(* Logix 5000 project; controller STAT 1756-L72 rev 20.12; software revision 20.04 *)

TASK IBT (periodic, rate 50 ms, priority 10, watchdog 200 ms) : ibt, stock, BASSIN
TASK MainTask (event, rate 200 ms, priority 15, watchdog 500 ms) : MainProgram

MODULES
   Local : 1756-L72 (ICP 0, rev 20.12)
        arm1_flex:0:I.1   // NIV_MID_VLOK1
        arm1_flex:0:I.2   // NIV_LAAG_VLOK1
        arm1_flex:0:I.4   // NIV_MID_VLOK2 FLOCULANT
        arm1_flex:0:I.5   // NIV_LAAG_VLOK2
        arm1_flex:0:I.6   // FC EV3
        arm1_flex:0:I.7   // FC EV3
        arm1_flex:0:I.12   // FLOW SWITCH PM4
        arm1_flex:0:I.13   // FLOW SWITCH PM2
        arm1_flex:0:I.14   // FLOW SWITCH PM3
        arm1_flex:0:I.15   // FLOW SWITCH PM4
        armstat_flex1:1:I.1   // CL3 MANU/AUTO
        armstat_flex1:4:O.0   // L P11 RUN
        armstat_flex1:4:O.1   // L P11 STOP/def
        armstat_flex1:4:O.2   // L P12 RUN
        armstat_flex1:4:O.3   // L P12 STOP/def
        armstat_flex1:4:O.4   // RES
        armstat_flex1:4:O.5   // RES
        armstat_flex1:4:O.6   // RES
        armstat_flex1:4:O.7   // RES
        armstat_flex1:4:O.8   // L P13 RUN
        armstat_flex1:4:O.9   // L P13 STOP/def
        armstat_flex1:4:O.10   // L P14 RUN
        armstat_flex1:4:O.11   // L P14 STOP/def
        armstat_flex1:4:O.12   // RES
        armstat_flex1:4:O.13   // RES
        armstat_flex1:4:O.14   // RES
        armstat_flex1:4:O.15   // RES
        armstat_flex1:0:I.1   // CL2 MANU/AUTO
        arm1_flex:1:I.0   // STFA11 EV1 BOVEN OPEN
        arm1_flex:1:I.1   // STFA11 EV1 BOVEN TOE
        arm1_flex:1:I.2   // STFA11 EV1 ONDER OPEN
        arm1_flex:1:I.3   // STFA11 EV1 ONDER TOE
        arm1_flex:1:I.4   // STFA12 EV1 BOVEN OPEN
        arm1_flex:1:I.5   // STFA12 EV1 BOVEN TOE
        arm1_flex:1:I.6   // STFA12 EV1 ONDER OPEN
        arm1_flex:1:I.7   // STFA12 EV1 ONDER TOE
        armstat_flex1:5:O.0   // L P15 RUN
        armstat_flex1:5:O.1   // L P15 STOP/def
        armstat_flex1:5:O.2   // L P16 RUN
        armstat_flex1:5:O.3   // L P16 STOP/def
        armstat_flex1:5:O.4   // RES
        armstat_flex1:5:O.5   // RES
        armstat_flex1:5:O.6   // RES
        armstat_flex1:5:O.7   // RES
        armstat_flex1:5:O.10   // RES
        armstat_flex1:5:O.11   // RES
        armstat_flex1:5:O.12   // RES
        armstat_flex1:5:O.13   // RES
        armstat_flex1:5:O.14   // RES
        armstat_flex1:5:O.15   // RES
        armstat_flex1:2:I.1   // CL4 MANU/AUTO
      usine : 1756-ENBT (Ethernet 192.168.3.162, ICP 1, rev 5.1)
         L1_usine : 1756-ENBT (Ethernet 192.168.3.159, rev 5.1)
            L1 : 1756-L72 (ICP 5, rev 20.1, $f88beb9a$ RPI 250 ms)
         EtherNet_Bridge : 1756-ENBT (Ethernet 192.168.3.150, rev 4.3)
            wkk : vendor 1 type 14 code 92 (ICP 2, rev 20.1, $435658c3$ RPI 20 ms)
         L2_usine : 1756-EN2T (Ethernet 192.168.3.163, rev 3.1)
            @63fa20a3@:Partner : vendor 1 type 14 code 146 (ICP 5, rev 20.1)
            L2PROCESS : vendor 1 type 14 code 147 (ICP 4, rev 20.1, $7ef97ec5$ RPI 20 ms)
         L3_usine : 1756-EN2T (Ethernet 192.168.3.161, rev 3.1)
            L3 : vendor 1 type 14 code 92 (ICP 0, rev 20.1, $abc03147$ RPI 250 ms)
      IO : 1756-ENBT (ICP 2, Ethernet 192.168.1.1, rev 6.4)
         arm1_flex : 1794-AENTR (Ethernet 192.168.1.8, rev 1.1, Output RPI 20 ms)
            I1_2 : 1794-IB16 (Flex 1, rev 1.1)
            I1_1 : 1794-IB16 (Flex 0, rev 1.1)
            I1_5 : 1794-IB16 (Flex 5, rev 1.1)
            O1_6 : vendor 1 type 7 code 35 (Flex 6, rev 1.1)
            N20 : vendor 1 type 10 code 31 (Flex 2, rev 1.1, Output RPI 80 ms)
            N21 : vendor 1 type 10 code 31 (Flex 3, rev 1.1, Output RPI 80 ms)
            N22 : vendor 1 type 10 code 31 (Flex 4, rev 1.1, Output RPI 80 ms)
         armstat_flex2 : 1794-AENTR (Ethernet 192.168.1.7, rev 1.1, Output RPI 20 ms)
            future : vendor 1 type 10 code 30 (Flex 1, rev 1.1, Input RPI 80 ms)
            N19_0 : vendor 1 type 10 code 30 (Flex 0, rev 1.1, Input RPI 80 ms)
         armPmp_flex1 : 1794-AENTR (Ethernet 192.168.1.5, rev 1.1, Output RPI 20 ms)
            I1_10 : 1794-IB16 (Flex 2, rev 1.1)
            I1_9 : 1794-IB16 (Flex 1, rev 1.1)
            O1_11 : vendor 1 type 7 code 35 (Flex 3, rev 1.1)
            I1_8 : 1794-IB16 (Flex 0, rev 1.1)
            O1_12 : vendor 1 type 7 code 35 (Flex 4, rev 1.1)
            N24 : vendor 1 type 10 code 31 (Flex 6, rev 1.1, Output RPI 80 ms)
            N23 : vendor 1 type 10 code 30 (Flex 5, rev 1.1, Input RPI 80 ms)
         armstat_flex1 : 1794-AENTR (Ethernet 192.168.1.6, rev 1.1, Output RPI 20 ms)
            I1_17 : 1794-IB16 (Flex 1, rev 1.1)
            O1_21 : vendor 1 type 7 code 35 (Flex 5, rev 1.1)
            I1_19 : 1794-IB16 (Flex 3, rev 1.1)
            I1_16 : 1794-IB16 (Flex 0, rev 1.1)
            I1_18 : 1794-IB16 (Flex 2, rev 1.1)
            O1_20 : vendor 1 type 7 code 35 (Flex 4, rev 1.1)
            N7_0 : vendor 1 type 10 code 30 (Flex 6, rev 1.1, Input RPI 80 ms)
         switch : vendor 1 type 12 code 238 (Ethernet 192.168.1.20, rev 3.1, StandardDataDriven RPI 1000 ms)
         bassin : vendor 1 type 12 code 228 (Ethernet 192.168.1.11, rev 1.1)
            bas_I_01 : vendor 1 type 116 code 6 (SLCChassis 1, rev 1.1, StandardDataDriven RPI 200 ms)
                 bassin:1:I.DATA.0   // fc vanne venturi ouverte vers venturi
                 bassin:1:I.DATA.1   // fc vanne venturi fermée vers bassin
                 bassin:1:I.DATA.2   // fc vanne PH bac ouverte
                 bassin:1:I.DATA.3   // fc vanne PH bac fermée
                 bassin:1:I.DATA.4   // fc vanne Neutral ouverte
                 bassin:1:I.DATA.5   // fc vanne Neutral fermée
                 bassin:1:I.DATA.6   // defaut ultima pmp renvoi 1
                 bassin:1:I.DATA.7   // defaut ultima pmp renvoi 2
                 bassin:1:I.DATA.8   // sélecteur local pmp renvoi 1
                 bassin:1:I.DATA.9   // Bp M/A loc pmp renvoi 1
                 bassin:1:I.DATA.10   // sélecteur local pmp renvoi 2
                 bassin:1:I.DATA.11   // Bp M/A loc pmp renvoi 2
                 bassin:1:I.DATA.12   // Bp M/A dist pmp renvoi 1
                 bassin:1:I.DATA.13   // Bp M/A dist pmp renvoi 2
                 bassin:1:I.DATA.14   // présence pmp renvoi 1
                 bassin:1:I.DATA.15   // présence pmp renvoi 2
                 bassin:1:I.DATA.16   // ready drive pmp acide nautral
                 bassin:1:I.DATA.17   // ready drive pmp base neutral
                 bassin:1:I.DATA.18   // selecteur fermer vanne
                 bassin:1:I.DATA.19   // reserve
                 bassin:1:I.DATA.20   // reserve
                 bassin:1:I.DATA.21   // reserve
                 bassin:1:I.DATA.22   // reserve
                 bassin:1:I.DATA.23   // reserve
                 bassin:1:I.DATA.24   // reserve
                 bassin:1:I.DATA.25   // reserve
                 bassin:1:I.DATA.26   // reserve
                 bassin:1:I.DATA.27   // reserve
                 bassin:1:I.DATA.28   // reserve
                 bassin:1:I.DATA.29   // reserve
                 bassin:1:I.DATA.30   // reserve
                 bassin:1:I.DATA.31   // reserve
            bas_AI_03 : vendor 1 type 117 code 6 (SLCChassis 3, rev 1.1, StandardDataDriven RPI 200 ms)
            bas_O_02 : vendor 1 type 116 code 30 (SLCChassis 2, rev 1.1, StandardDataDriven RPI 200 ms)
                 bassin:2:O.POINT_11   // pmp acide
                 bassin:2:O.POINT_12   // ajout base
                 bassin:2:O.DATA.0   // marche pmp 1 renvoi
                 bassin:2:O.DATA.1   // marche pmp 2 renvoi
                 bassin:2:O.DATA.2   // ouverturre vanne venturi
                 bassin:2:O.DATA.3   // lampe M/A loc pmp renvoi 1
                 bassin:2:O.DATA.4   // lampe M/A loc pmp renvoi 2
                 bassin:2:O.DATA.5   // lampe M/A dist pmp renvoi 1
                 bassin:2:O.DATA.6   // lampe M/A dist pmp renvoi 2
                 bassin:2:O.DATA.7   // colone lumineuse bleu discord. vanne manu
                 bassin:2:O.DATA.8   // colone lumineuse niveau bas bassin
                 bassin:2:O.DATA.9   // colone lumineuse defaut pompe renvoi
                 bassin:2:O.DATA.10   // colone lumineuse rouge
                 bassin:2:O.DATA.11   // M/A drive PMP acide neutral
                 bassin:2:O.DATA.12   // M/A drive PMP base neutral
                 bassin:2:O.DATA.13   // reserve
                 bassin:2:O.DATA.14   // reserve
                 bassin:2:O.DATA.15   // reserve
                 bassin:2:O.DATA.16   // reserve
                 bassin:2:O.DATA.17   // reserve
                 bassin:2:O.DATA.18   // reserve
                 bassin:2:O.DATA.19   // reserve
                 bassin:2:O.DATA.20   // reserve
                 bassin:2:O.DATA.21   // reserve
                 bassin:2:O.DATA.22   // reserve
                 bassin:2:O.DATA.23   // reserve
                 bassin:2:O.DATA.24   // reserve
                 bassin:2:O.DATA.25   // reserve
                 bassin:2:O.DATA.26   // reserve
                 bassin:2:O.DATA.27   // reserve
                 bassin:2:O.DATA.28   // reserve
                 bassin:2:O.DATA.29   // reserve
                 bassin:2:O.DATA.30   // reserve
                 bassin:2:O.DATA.31   // reserve
            bas_AO_04 : vendor 1 type 117 code 11 (SLCChassis 4, rev 1.1, StandardDataDriven RPI 200 ms)
                 bassin:4:O.CHANNEL_0_OUTPUT   // consigne position vanne renvoi
                 bassin:4:O.CHANNEL_1_OUTPUT   // consigne vitesse pmp acide neutral
                 bassin:4:O.CHANNEL_2_OUTPUT   // consigne vitesse pmp base neutral
         Lancy_R2 : vendor 1 type 12 code 228 (Ethernet 192.168.1.14, rev 1.1)
            lancy_R2_O2 : vendor 1 type 116 code 23 (SLCChassis 2, rev 1.1, StandardDataDriven RPI 200 ms)
                 Lancy_R2:2:O.DATA.0   // drum wash frequency. duration timer panel+G116
                 Lancy_R2:2:O.DATA.1   // surge tank T150 overflow shut off valve
                 Lancy_R2:2:O.DATA.2   // AV 147 open
                 Lancy_R2:2:O.DATA.3   // AV 147 close
                 Lancy_R2:2:O.DATA.4   // caustic supply P190
                 Lancy_R2:2:O.DATA.5   // P190 on
                 Lancy_R2:2:O.DATA.6   // ST VA7 Vanne eau rinçage
                 Lancy_R2:2:O.DATA.7   // ST VA7 Vanne eau rinçage
                 Lancy_R2:2:O.POINT_0   // drum wash frequency. duration timer panel+G116
                 Lancy_R2:2:O.POINT_1   // surge tank T150 overflow shut off valve
                 Lancy_R2:2:O.POINT_2   // AV 147 open
                 Lancy_R2:2:O.POINT_3   // AV 147 close
                 Lancy_R2:2:O.POINT_4   // caustic supply P190
                 Lancy_R2:2:O.POINT_5   // P190 on
                 Lancy_R2:2:O.POINT_6   // ST VA7 Vanne eau rinçage
                 Lancy_R2:2:O.POINT_7   // ST VA7 Vanne eau rinçage
            lancy_R2_O6 : vendor 1 type 116 code 23 (SLCChassis 6, rev 1.1, StandardDataDriven RPI 200 ms)
                 Lancy_R2:6:O.DATA.0   // AV 330 closed
                 Lancy_R2:6:O.DATA.1   // alarm horn
                 Lancy_R2:6:O.DATA.2   // L1 high level
                 Lancy_R2:6:O.DATA.3   // L1 low level
                 Lancy_R2:6:O.DATA.4   // L2 high level
                 Lancy_R2:6:O.DATA.5   // L2 low level
                 Lancy_R2:6:O.DATA.6   // L3 high level
                 Lancy_R2:6:O.DATA.7   // L3 low level
                 Lancy_R2:6:O.POINT_0   // AV 330 closed
                 Lancy_R2:6:O.POINT_1   // alarm horn
                 Lancy_R2:6:O.POINT_2   // L1 high level
                 Lancy_R2:6:O.POINT_3   // L1 low level
                 Lancy_R2:6:O.POINT_4   // L2 high level
                 Lancy_R2:6:O.POINT_5   // L2 low level
                 Lancy_R2:6:O.POINT_6   // L3 high level
                 Lancy_R2:6:O.POINT_7   // L3 low level
            lancy_R2_O9 : vendor 1 type 116 code 23 (SLCChassis 9, rev 1.1, StandardDataDriven RPI 200 ms)
                 Lancy_R2:9:O.DATA.0   // cloudy filtrate P240 overcurrent
                 Lancy_R2:9:O.DATA.1   // rotary drum F200 overcurrent
                 Lancy_R2:9:O.DATA.2   // vacuum pump P250 overcurrent
                 Lancy_R2:9:O.DATA.3   // clear filtrate pump failure
                 Lancy_R2:9:O.DATA.4   // cloudy filtrate pump failure
                 Lancy_R2:9:O.DATA.5   // filtrate lift station pump failure
                 Lancy_R2:9:O.DATA.6   // regenerate caustic avalaible holding tank
                 Lancy_R2:9:O.DATA.7   // System high level alarm
                 Lancy_R2:9:O.POINT_0   // cloudy filtrate P240 overcurrent
                 Lancy_R2:9:O.POINT_1   // rotary drum F200 overcurrent
                 Lancy_R2:9:O.POINT_2   // vacuum pump P250 overcurrent
                 Lancy_R2:9:O.POINT_3   // clear filtrate pump failure
                 Lancy_R2:9:O.POINT_4   // cloudy filtrate pump failure
                 Lancy_R2:9:O.POINT_5   // filtrate lift station pump failure
                 Lancy_R2:9:O.POINT_6   // regenerate caustic avalaible holding tank
                 Lancy_R2:9:O.POINT_7   // System high level alarm
            lancy_R2_O7 : vendor 1 type 116 code 23 (SLCChassis 7, rev 1.1, StandardDataDriven RPI 200 ms)
                 Lancy_R2:7:O.DATA.0   // holding tank T130 high level
                 Lancy_R2:7:O.DATA.1   // filtrate lift station T160 high level
                 Lancy_R2:7:O.DATA.2   // clear filtrate receiver T260 high level
                 Lancy_R2:7:O.DATA.3   // cloudy filtrate receiver T270 high level
                 Lancy_R2:7:O.DATA.4   // vacuum pump sunction line high level
                 Lancy_R2:7:O.DATA.5   // reactor tank T100 high level
                 Lancy_R2:7:O.DATA.6   // reactor tank T100 low level
                 Lancy_R2:7:O.DATA.7   // vacuum pump P250 seal water low flow
                 Lancy_R2:7:O.POINT_0   // holding tank T130 high level
                 Lancy_R2:7:O.POINT_1   // filtrate lift station T160 high level
                 Lancy_R2:7:O.POINT_2   // clear filtrate receiver T260 high level
                 Lancy_R2:7:O.POINT_3   // cloudy filtrate receiver T270 high level
                 Lancy_R2:7:O.POINT_4   // vacuum pump sunction line high level
                 Lancy_R2:7:O.POINT_5   // reactor tank T100 high level
                 Lancy_R2:7:O.POINT_6   // reactor tank T100 low level
                 Lancy_R2:7:O.POINT_7   // vacuum pump P250 seal water low flow
            lancy_R2_O4 : vendor 1 type 116 code 23 (SLCChassis 4, rev 1.1, StandardDataDriven RPI 200 ms)
                 Lancy_R2:4:O.DATA.0   // LV 315 open
                 Lancy_R2:4:O.DATA.1   // LV 315 closed
                 Lancy_R2:4:O.DATA.2   // L2 filtrate return valve
                 Lancy_R2:4:O.DATA.3   // LV 325 open
                 Lancy_R2:4:O.DATA.4   // LV 325 closed
                 Lancy_R2:4:O.DATA.5   // L1 filtrate return valve
                 Lancy_R2:4:O.DATA.6   // LV 335 open
                 Lancy_R2:4:O.DATA.7   // LV 335 closed
                 Lancy_R2:4:O.POINT_0   // LV 315 open
                 Lancy_R2:4:O.POINT_1   // LV 315 closed
                 Lancy_R2:4:O.POINT_2   // L2 filtrate return valve
                 Lancy_R2:4:O.POINT_3   // LV 325 open
                 Lancy_R2:4:O.POINT_4   // LV 325 closed
                 Lancy_R2:4:O.POINT_5   // L1 filtrate return valve
                 Lancy_R2:4:O.POINT_6   // LV 335 open
                 Lancy_R2:4:O.POINT_7   // LV 335 closed
            lancy_R2_O3 : vendor 1 type 116 code 23 (SLCChassis 3, rev 1.1, StandardDataDriven RPI 200 ms)
                 Lancy_R2:3:O.DATA.0   // res
                 Lancy_R2:3:O.DATA.1   // L4 reactor return valve
                 Lancy_R2:3:O.DATA.2   // LV 420 open
                 Lancy_R2:3:O.DATA.3   // LV 420 closed
                 Lancy_R2:3:O.DATA.4   // run pompe op008
                 Lancy_R2:3:O.DATA.5   // L4 high level
                 Lancy_R2:3:O.DATA.6   // L4 low level
                 Lancy_R2:3:O.DATA.7   // L3 filtrate return valve
                 Lancy_R2:3:O.POINT_0   // res
                 Lancy_R2:3:O.POINT_1   // L4 reactor return valve
                 Lancy_R2:3:O.POINT_2   // LV 420 open
                 Lancy_R2:3:O.POINT_3   // LV 420 closed
                 Lancy_R2:3:O.POINT_4   // run pompe op008
                 Lancy_R2:3:O.POINT_5   // L4 high level
                 Lancy_R2:3:O.POINT_6   // L4 low level
                 Lancy_R2:3:O.POINT_7   // L3 filtrate return valve
            lancy_R2_O5 : vendor 1 type 116 code 23 (SLCChassis 5, rev 1.1, StandardDataDriven RPI 200 ms)
                 Lancy_R2:5:O.DATA.0   // reactor return flow valve AV 310
                 Lancy_R2:5:O.DATA.1   // AV 310 open
                 Lancy_R2:5:O.DATA.2   // AV 310 closed
                 Lancy_R2:5:O.DATA.3   // reactor return flow valve AV 320
                 Lancy_R2:5:O.DATA.4   // AV 320 open
                 Lancy_R2:5:O.DATA.5   // AV 320 closed
                 Lancy_R2:5:O.DATA.6   // reactor return flow valve AV 330
                 Lancy_R2:5:O.DATA.7   // AV 330 open
                 Lancy_R2:5:O.POINT_0   // reactor return flow valve AV 310
                 Lancy_R2:5:O.POINT_1   // AV 310 open
                 Lancy_R2:5:O.POINT_2   // AV 310 closed
                 Lancy_R2:5:O.POINT_3   // reactor return flow valve AV 320
                 Lancy_R2:5:O.POINT_4   // AV 320 open
                 Lancy_R2:5:O.POINT_5   // AV 320 closed
                 Lancy_R2:5:O.POINT_6   // reactor return flow valve AV 330
                 Lancy_R2:5:O.POINT_7   // AV 330 open
            lancy_R2_O1 : vendor 1 type 116 code 23 (SLCChassis 1, rev 1.1, StandardDataDriven RPI 200 ms)
                 Lancy_R2:1:O.DATA.0   // vacuum pump P250 seal water valve
                 Lancy_R2:1:O.DATA.1   // reactor tank mixer M120 (15,16,17,990)
                 Lancy_R2:1:O.DATA.2   // M120 run
                 Lancy_R2:1:O.DATA.3   // M110 run speed control operation
                 Lancy_R2:1:O.DATA.4   // M110 run bypass
                 Lancy_R2:1:O.DATA.5   // rotary drum vacuum filter F200 (50,51,52,984)
                 Lancy_R2:1:O.DATA.6   // F200 run
                 Lancy_R2:1:O.DATA.7   // reserve
                 Lancy_R2:1:O.POINT_0   // vacuum pump P250 seal water valve
                 Lancy_R2:1:O.POINT_1   // reactor tank mixer M120 (15,16,17,990)
                 Lancy_R2:1:O.POINT_2   // M120 run
                 Lancy_R2:1:O.POINT_3   // M110 run speed control operation
                 Lancy_R2:1:O.POINT_4   // M110 run bypass
                 Lancy_R2:1:O.POINT_5   // rotary drum vacuum filter F200 (50,51,52,984)
                 Lancy_R2:1:O.POINT_6   // F200 run
                 Lancy_R2:1:O.POINT_7   // reserve
            lancy_R2_O8 : vendor 1 type 116 code 23 (SLCChassis 8, rev 1.1, StandardDataDriven RPI 200 ms)
                 Lancy_R2:8:O.DATA.0   // surge tank T150 high turbidity
                 Lancy_R2:8:O.DATA.1   // slury mixer M110 failure
                 Lancy_R2:8:O.DATA.2   // shearing mixer M120 overcurrent
                 Lancy_R2:8:O.DATA.3   // filtrate pump P170 overcurrent
                 Lancy_R2:8:O.DATA.4   // filtrate pump P180 overcurrent
                 Lancy_R2:8:O.DATA.5   // clear filtrate P210 overcurrent
                 Lancy_R2:8:O.DATA.6   // clear filtrate P220 overcurrent
                 Lancy_R2:8:O.DATA.7   // cloudy filtrate P230 overcurrent
                 Lancy_R2:8:O.POINT_0   // surge tank T150 high turbidity
                 Lancy_R2:8:O.POINT_1   // slury mixer M110 failure
                 Lancy_R2:8:O.POINT_2   // shearing mixer M120 overcurrent
                 Lancy_R2:8:O.POINT_3   // filtrate pump P170 overcurrent
                 Lancy_R2:8:O.POINT_4   // filtrate pump P180 overcurrent
                 Lancy_R2:8:O.POINT_5   // clear filtrate P210 overcurrent
                 Lancy_R2:8:O.POINT_6   // clear filtrate P220 overcurrent
                 Lancy_R2:8:O.POINT_7   // cloudy filtrate P230 overcurrent
         Lancy_R3 : vendor 1 type 12 code 228 (Ethernet 192.168.1.15, rev 1.1)
            lancy_R3_AI8 : vendor 1 type 117 code 6 (SLCChassis 8, rev 1.1, StandardDataDriven RPI 200 ms)
                 Lancy_R3:8:I.CHANNEL_0_DATA   // op008
                 Lancy_R3:8:I.CHANNEL_1_DATA   // op009
                 Lancy_R3:8:I.CHANNEL_2_DATA   // op010
                 Lancy_R3:8:I.CHANNEL_3_DATA   // op011
                 Lancy_R3:8:I.CHANNEL_4_DATA   // op007
                 Lancy_R3:8:I.CHANNEL_5_DATA   // op006
                 Lancy_R3:8:I.CHANNEL_6_DATA   // stock soude pellet L4
                 Lancy_R3:8:I.CHANNEL_7_DATA   // reserve
            lancy_R3_AO5 : vendor 1 type 117 code 11 (SLCChassis 5, rev 1.1, StandardDataDriven RPI 200 ms)
                 Lancy_R3:5:O.CHANNEL_0_OUTPUT   // sortie analog position servo vanne filtrat de 0 à 200
                 Lancy_R3:5:O.CHANNEL_1_OUTPUT   // reserve
                 Lancy_R3:5:O.CHANNEL_2_OUTPUT   // reserve
                 Lancy_R3:5:O.CHANNEL_3_OUTPUT   // reserve
            lancy_R3_O1 : vendor 1 type 116 code 23 (SLCChassis 1, rev 1.1, StandardDataDriven RPI 200 ms)
                 Lancy_R3:1:O.DATA.0   // reactor tank T100 water make up valve LV 346
                 Lancy_R3:1:O.DATA.1   // LV 346 open
                 Lancy_R3:1:O.DATA.2   // LV 346 closed
                 Lancy_R3:1:O.DATA.3   // System high high alarm
                 Lancy_R3:1:O.DATA.4   // vanne stock soude
                 Lancy_R3:1:O.DATA.5   // vanne soude bouilloire
                 Lancy_R3:1:O.DATA.6   // klaxon niveau stock
                 Lancy_R3:1:O.DATA.7   // lampe niveau stock
                 Lancy_R3:1:O.POINT_0   // reactor tank T100 water make up valve LV 346
                 Lancy_R3:1:O.POINT_1   // LV 346 open
                 Lancy_R3:1:O.POINT_2   // LV 346 closed
                 Lancy_R3:1:O.POINT_3   // System high high alarm
                 Lancy_R3:1:O.POINT_4   // vanne stock soude
                 Lancy_R3:1:O.POINT_5   // vanne soude bouilloire
                 Lancy_R3:1:O.POINT_6   // klaxon niveau stock
                 Lancy_R3:1:O.POINT_7   // lampe niveau stock
            lancy_R3_I2 : vendor 1 type 116 code 12 (SLCChassis 2, rev 1.1, StandardDataDriven RPI 200 ms)
                 Lancy_R3:2:I.DATA.0   // ST VA1 OPEN
                 Lancy_R3:2:I.DATA.1   // ST VA1 CLOSE
                 Lancy_R3:2:I.DATA.2   // ST VA2 OPEN
                 Lancy_R3:2:I.DATA.3   // ST VA2 CLOSE
                 Lancy_R3:2:I.DATA.4   // ST VA3 OPEN
                 Lancy_R3:2:I.DATA.5   // ST VA3 CLOSE
                 Lancy_R3:2:I.DATA.6   // ST VA4 OPEN
                 Lancy_R3:2:I.DATA.7   // ST VA4 CLOSE
                 Lancy_R3:2:I.DATA.8   // ST VA5 OPEN
                 Lancy_R3:2:I.DATA.9   // ST VA5 CLOSE
                 Lancy_R3:2:I.DATA.10   // ST VA6 OPEN
                 Lancy_R3:2:I.DATA.11   // ST VA6 CLOSE
                 Lancy_R3:2:I.DATA.12   // ST VA7 OPEN
                 Lancy_R3:2:I.DATA.13   // ST VA7 CLOSE
                 Lancy_R3:2:I.DATA.14   // protection pompe eto op008
                 Lancy_R3:2:I.DATA.15   // reserve
                 Lancy_R3:2:I.POINT_0   // ST VA1 OPEN
                 Lancy_R3:2:I.POINT_1   // ST VA1 CLOSE
                 Lancy_R3:2:I.POINT_2   // ST VA2 OPEN
                 Lancy_R3:2:I.POINT_3   // ST VA2 CLOSE
                 Lancy_R3:2:I.POINT_4   // ST VA3 OPEN
                 Lancy_R3:2:I.POINT_5   // ST VA3 CLOSE
                 Lancy_R3:2:I.POINT_6   // ST VA4 OPEN
                 Lancy_R3:2:I.POINT_7   // ST VA4 CLOSE
                 Lancy_R3:2:I.POINT_8   // ST VA5 OPEN
                 Lancy_R3:2:I.POINT_9   // ST VA5 CLOSE
                 Lancy_R3:2:I.POINT_10   // ST VA6 OPEN
                 Lancy_R3:2:I.POINT_11   // ST VA6 CLOSE
                 Lancy_R3:2:I.POINT_12   // ST VA7 OPEN
                 Lancy_R3:2:I.POINT_13   // ST VA7 CLOSE
                 Lancy_R3:2:I.POINT_14   // protection pompe eto op008
                 Lancy_R3:2:I.POINT_15   // level hcl
            lancy_R3_O3 : vendor 1 type 116 code 23 (SLCChassis 3, rev 1.1, StandardDataDriven RPI 200 ms)
                 Lancy_R3:3:O.DATA.0   // marche pmp 1 puisard L123
                 Lancy_R3:3:O.DATA.1   // marche pmp 2 puisard L123
                 Lancy_R3:3:O.DATA.2   // ST VA1 vanne remplissage OP008
                 Lancy_R3:3:O.DATA.3   // ST VA2 vanne aspiration PP1 OP008
                 Lancy_R3:3:O.DATA.4   // ST VA3
                 Lancy_R3:3:O.DATA.5   // ST VA4 vanne holding tank
                 Lancy_R3:3:O.DATA.6   // ST VA5 vanne reactor
                 Lancy_R3:3:O.DATA.7   // ST VA6 vers L4
                 Lancy_R3:3:O.POINT_0   // marche pmp 1 puisard L123
                 Lancy_R3:3:O.POINT_1   // marche pmp 2 puisard L123
                 Lancy_R3:3:O.POINT_2   // ST VA1 vanne remplissage OP008
                 Lancy_R3:3:O.POINT_3   // ST VA2 vanne aspiration PP1 OP008
                 Lancy_R3:3:O.POINT_4   // ST VA3
                 Lancy_R3:3:O.POINT_5   // ST VA4 vanne holding tank
                 Lancy_R3:3:O.POINT_6   // ST VA5 vanne reactor
                 Lancy_R3:3:O.POINT_7   // ST VA6 vers L4
            lancy_R3_AI4 : vendor 1 type 117 code 6 (SLCChassis 4, rev 1.1, StandardDataDriven RPI 200 ms)
                 Lancy_R3:4:I.CHANNEL_0_DATA   // flow filter presse
                 Lancy_R3:4:I.CHANNEL_1_DATA   // pos valve filtrat
                 Lancy_R3:4:I.CHANNEL_2_DATA   // niveau reacteur
                 Lancy_R3:4:I.CHANNEL_3_DATA   // reserve
                 Lancy_R3:4:I.CHANNEL_4_DATA   // hac turbidity
                 Lancy_R3:4:I.CHANNEL_5_DATA   // optek turbidity
                 Lancy_R3:4:I.CHANNEL_6_DATA   // niveau BUFFER VOOR FILTER PERS
                 Lancy_R3:4:I.CHANNEL_7_DATA   // LEVEL FLITRAAT WATER FROM FILTERPERS
            lancy_R3_AI6 : vendor 1 type 117 code 6 (SLCChassis 6, rev 1.1, StandardDataDriven RPI 200 ms)
                 Lancy_R3:6:I.CHANNEL_0_DATA   // flow naoh from L1
                 Lancy_R3:6:I.CHANNEL_1_DATA   // flow naoh from L2
                 Lancy_R3:6:I.CHANNEL_2_DATA   // flow naoh from L3
                 Lancy_R3:6:I.CHANNEL_3_DATA   // level holding tank
                 Lancy_R3:6:I.CHANNEL_4_DATA   // level lift tank
                 Lancy_R3:6:I.CHANNEL_5_DATA   // reserve
                 Lancy_R3:6:I.CHANNEL_6_DATA   // reserve
                 Lancy_R3:6:I.CHANNEL_7_DATA   // reserve
                 Lancy_R3:6:I.CHANNEL_0_STATUS   // reserve
            lancy_R3_AO7 : vendor 1 type 117 code 11 (SLCChassis 7, rev 1.1, StandardDataDriven RPI 200 ms)
                 Lancy_R3:7:O.CHANNEL_0_OUTPUT   // AFFICHEUR DEBIT L1
                 Lancy_R3:7:O.CHANNEL_1_OUTPUT   // AFFICHEUR DEBIT L2
                 Lancy_R3:7:O.CHANNEL_2_OUTPUT   // AFFICHEUR DEBIT L3
                 Lancy_R3:7:O.CHANNEL_3_OUTPUT   // AFFICHEUR TOTAL DEBIt
         stock : vendor 1 type 12 code 228 (Ethernet 192.168.1.13, rev 1.1)
            stock_I1 : vendor 1 type 116 code 6 (SLCChassis 1, rev 1.1, StandardDataDriven RPI 20 ms)
            stock_I4 : vendor 1 type 117 code 6 (SLCChassis 4, rev 1.1, StandardDataDriven RPI 20 ms)
            stock_I2 : vendor 1 type 116 code 6 (SLCChassis 2, rev 1.1, StandardDataDriven RPI 20 ms)
                 stock:2:I.DATA.23   // pulse gaz chaud L3
                 stock:2:I.POINT_23   // pulse gaz chaud L3 1m³/pulse
            stock_O3 : vendor 1 type 116 code 30 (SLCChassis 3, rev 1.1, StandardDataDriven RPI 20 ms)
            O6 : vendor 1 type 116 code 30 (SLCChassis 6, rev 1.1, StandardDataDriven RPI 20 ms)
            stock_I5 : vendor 1 type 117 code 6 (SLCChassis 5, rev 1.1, StandardDataDriven RPI 20 ms)
         Lancy_R1 : vendor 1 type 12 code 228 (Ethernet 192.168.1.10, rev 1.1)
            lancy_R1_I7 : vendor 1 type 116 code 12 (SLCChassis 7, rev 1.1, StandardDataDriven RPI 200 ms)
                 Lancy_R1:7:I.DATA.0   // P220 overcurrent
                 Lancy_R1:7:I.DATA.1   // P230 overcurrent
                 Lancy_R1:7:I.DATA.2   // P240 overcurrent
                 Lancy_R1:7:I.DATA.3   // F200 overcurrent
                 Lancy_R1:7:I.DATA.4   // P250 overcurrent
                 Lancy_R1:7:I.DATA.5   // L4 level point LE 400 A
                 Lancy_R1:7:I.DATA.6   // L4 level point LE 400 B
                 Lancy_R1:7:I.DATA.7   // L4 level point LE 400 C
                 Lancy_R1:7:I.DATA.8   // reactor tank T100 LE 106 E low level alarm
                 Lancy_R1:7:I.DATA.9   // reactor tank T100 water make up valve LV 346 auto
                 Lancy_R1:7:I.DATA.10   // reactor tank T100 water make up valve LV 346 close
                 Lancy_R1:7:I.DATA.11   // holding tank T130 level point LE 135 B
                 Lancy_R1:7:I.DATA.12   // L4 level point LE 400 D
                 Lancy_R1:7:I.DATA.13   // L4 level point LE 400 E
                 Lancy_R1:7:I.DATA.14   // mixer defaut phase
                 Lancy_R1:7:I.DATA.15   // reserve
                 Lancy_R1:7:I.POINT_0   // P220 overcurrent
                 Lancy_R1:7:I.POINT_1   // P230 overcurrent
                 Lancy_R1:7:I.POINT_2   // P240 overcurrent
                 Lancy_R1:7:I.POINT_3   // F200 overcurrent
                 Lancy_R1:7:I.POINT_4   // P250 overcurrent
                 Lancy_R1:7:I.POINT_5   // L4 level point LE 400 A
                 Lancy_R1:7:I.POINT_6   // L4 level point LE 400 B
                 Lancy_R1:7:I.POINT_7   // L4 level point LE 400 C
                 Lancy_R1:7:I.POINT_8   // reactor tank T100 LE 106 E low level alarm
                 Lancy_R1:7:I.POINT_9   // reactor tank T100 water make up valve LV 346 auto
                 Lancy_R1:7:I.POINT_10   // reactor tank T100 water make up valve LV 346 close
                 Lancy_R1:7:I.POINT_11   // holding tank T130 level point LE 135 B
                 Lancy_R1:7:I.POINT_12   // L4 level point LE 400 D
                 Lancy_R1:7:I.POINT_13   // L4 level point LE 400 E
                 Lancy_R1:7:I.POINT_14   // mixer defaut phase
                 Lancy_R1:7:I.POINT_15   // reserve
            lancy_R1_I2 : vendor 1 type 116 code 12 (SLCChassis 2, rev 1.1, StandardDataDriven RPI 200 ms)
                 Lancy_R1:2:I.DATA.0   // fc vanne bouilloire open
                 Lancy_R1:2:I.DATA.1   // fc vanne bouilloire closed
                 Lancy_R1:2:I.DATA.2   // bp open vanne silo
                 Lancy_R1:2:I.DATA.3   // bp open vanne bouilloire
                 Lancy_R1:2:I.DATA.4   // holding tank T130 LE135 A
                 Lancy_R1:2:I.DATA.5   // filtrate lift station T160 LE165 A
                 Lancy_R1:2:I.DATA.6   // filtrate lift station T160 LE165 B
                 Lancy_R1:2:I.DATA.7   // filtrate lift station T160 LE165 C
                 Lancy_R1:2:I.DATA.8   // filtrate lift station T160 LE165 D
                 Lancy_R1:2:I.DATA.9   // clear filtrate receiver T260 LE265
                 Lancy_R1:2:I.DATA.10   // cloudy filtrate receiver T270 LE275
                 Lancy_R1:2:I.DATA.11   // vacuum pump suction line LE285
                 Lancy_R1:2:I.DATA.12   // reactor tank T100 LE106 A
                 Lancy_R1:2:I.DATA.13   // reactor tank T100 LE106 B
                 Lancy_R1:2:I.DATA.14   // reactor tank T100 LE106 C
                 Lancy_R1:2:I.DATA.15   // reactor tank T100 LE106 D
                 Lancy_R1:2:I.POINT_0   // fc vanne bouilloire open
                 Lancy_R1:2:I.POINT_1   // fc vanne bouilloire closed
                 Lancy_R1:2:I.POINT_2   // bp open vanne silo
                 Lancy_R1:2:I.POINT_3   // bp open vanne bouilloire
                 Lancy_R1:2:I.POINT_4   // holding tank T130 LE135 A
                 Lancy_R1:2:I.POINT_5   // filtrate lift station T160 LE165 A
                 Lancy_R1:2:I.POINT_6   // filtrate lift station T160 LE165 B
                 Lancy_R1:2:I.POINT_7   // filtrate lift station T160 LE165 C
                 Lancy_R1:2:I.POINT_8   // filtrate lift station T160 LE165 D
                 Lancy_R1:2:I.POINT_9   // clear filtrate receiver T260 LE265
                 Lancy_R1:2:I.POINT_10   // cloudy filtrate receiver T270 LE275
                 Lancy_R1:2:I.POINT_11   // vacuum pump suction line LE285
                 Lancy_R1:2:I.POINT_12   // reactor tank T100 LE106 A
                 Lancy_R1:2:I.POINT_13   // reactor tank T100 LE106 B
                 Lancy_R1:2:I.POINT_14   // reactor tank T100 LE106 C
                 Lancy_R1:2:I.POINT_15   // reactor tank T100 LE106 D
            lancy_R1_I5 : vendor 1 type 116 code 12 (SLCChassis 5, rev 1.1, StandardDataDriven RPI 200 ms)
                 Lancy_R1:5:I.DATA.0   // HS 110 off
                 Lancy_R1:5:I.DATA.1   // M110 run speed controller operation
                 Lancy_R1:5:I.DATA.2   // M110 overcurrent
                 Lancy_R1:5:I.DATA.3   // auto surge tank T150 overflow shut off valve AV147
                 Lancy_R1:5:I.DATA.4   // man surge tank T150 overflow shut off valve AV147
                 Lancy_R1:5:I.DATA.5   // auto caustic supply P190
                 Lancy_R1:5:I.DATA.6   // man caustic supply P190
                 Lancy_R1:5:I.DATA.7   // caustic batching controller rub caustic pump P190
                 Lancy_R1:5:I.DATA.8   // auto L4 filtrate return valve LV410
                 Lancy_R1:5:I.DATA.9   // open L4 filtrate return valve LV410
                 Lancy_R1:5:I.DATA.10   // auto L4 reactor return valve AV420
                 Lancy_R1:5:I.DATA.11   // close L4 reactor return valve AV420
                 Lancy_R1:5:I.DATA.12   // reserve
                 Lancy_R1:5:I.DATA.13   // reserve
                 Lancy_R1:5:I.DATA.14   // auto L3 filtrate return valve LV315
                 Lancy_R1:5:I.DATA.15   // open L3 filtrate return valve LV315
                 Lancy_R1:5:I.POINT_0   // HS 110 off
                 Lancy_R1:5:I.POINT_1   // M110 run speed controller operation
                 Lancy_R1:5:I.POINT_2   // M110 overcurrent
                 Lancy_R1:5:I.POINT_3   // auto surge tank T150 overflow shut off valve AV147
                 Lancy_R1:5:I.POINT_4   // man surge tank T150 overflow shut off valve AV147
                 Lancy_R1:5:I.POINT_5   // auto caustic supply P190
                 Lancy_R1:5:I.POINT_6   // man caustic supply P190
                 Lancy_R1:5:I.POINT_7   // caustic batching controller rub caustic pump P190
                 Lancy_R1:5:I.POINT_8   // auto L4 filtrate return valve LV410
                 Lancy_R1:5:I.POINT_9   // open L4 filtrate return valve LV410
                 Lancy_R1:5:I.POINT_10   // auto L4 reactor return valve AV420
                 Lancy_R1:5:I.POINT_11   // close L4 reactor return valve AV420
                 Lancy_R1:5:I.POINT_12   // reserve
                 Lancy_R1:5:I.POINT_13   // reserve
                 Lancy_R1:5:I.POINT_14   // auto L3 filtrate return valve LV315
                 Lancy_R1:5:I.POINT_15   // open L3 filtrate return valve LV315
            lancy_R1_I1 : vendor 1 type 116 code 12 (SLCChassis 1, rev 1.1, StandardDataDriven RPI 200 ms)
                 Lancy_R1:1:I.DATA.0   // master control relay
                 Lancy_R1:1:I.DATA.1   // acknowledge alarm
                 Lancy_R1:1:I.DATA.2   // reset alarm
                 Lancy_R1:1:I.DATA.3   // test alarm
                 Lancy_R1:1:I.DATA.4   // test lamps
                 Lancy_R1:1:I.DATA.5   // L1 level point LE337 A
                 Lancy_R1:1:I.DATA.6   // L1 level point LE337 B
                 Lancy_R1:1:I.DATA.7   // L1 level point LE337 C
                 Lancy_R1:1:I.DATA.8   // L1 level point LE337 D
                 Lancy_R1:1:I.DATA.9   // L1 level point LE337 E
                 Lancy_R1:1:I.DATA.10   // L2 level point LE327 A
                 Lancy_R1:1:I.DATA.11   // L2 level point LE327 B
                 Lancy_R1:1:I.DATA.12   // L2 level point LE327 C
                 Lancy_R1:1:I.DATA.13   // L2 level point LE327 D
                 Lancy_R1:1:I.DATA.14   // fc vanne silo open
                 Lancy_R1:1:I.DATA.15   // fc vanne silo closed
                 Lancy_R1:1:I.POINT_0   // master control relay
                 Lancy_R1:1:I.POINT_1   // acknowledge alarm
                 Lancy_R1:1:I.POINT_2   // reset alarm
                 Lancy_R1:1:I.POINT_3   // test alarm
                 Lancy_R1:1:I.POINT_4   // test lamps
                 Lancy_R1:1:I.POINT_5   // L1 level point LE337 A
                 Lancy_R1:1:I.POINT_6   // L1 level point LE337 B
                 Lancy_R1:1:I.POINT_7   // L1 level point LE337 C
                 Lancy_R1:1:I.POINT_8   // L1 level point LE337 D
                 Lancy_R1:1:I.POINT_9   // L1 level point LE337 E
                 Lancy_R1:1:I.POINT_10   // L2 level point LE327 A
                 Lancy_R1:1:I.POINT_11   // L2 level point LE327 B
                 Lancy_R1:1:I.POINT_12   // L2 level point LE327 C
                 Lancy_R1:1:I.POINT_13   // L2 level point LE327 D
                 Lancy_R1:1:I.POINT_14   // fc vanne silo open
                 Lancy_R1:1:I.POINT_15   // fc vanne silo closed
            lancy_R1_I4 : vendor 1 type 116 code 12 (SLCChassis 4, rev 1.1, StandardDataDriven RPI 200 ms)
                 Lancy_R1:4:I.DATA.0   // auto filtrate lift station P170
                 Lancy_R1:4:I.DATA.1   // man filtrate lift station P170
                 Lancy_R1:4:I.DATA.2   // P170 run
                 Lancy_R1:4:I.DATA.3   // auto filtrate lift station P180
                 Lancy_R1:4:I.DATA.4   // man filtrate lift station P180
                 Lancy_R1:4:I.DATA.5   // P180 run
                 Lancy_R1:4:I.DATA.6   // on clear filtrate P210
                 Lancy_R1:4:I.DATA.7   // Stand by clear filtrate P210
                 Lancy_R1:4:I.DATA.8   // P210 run
                 Lancy_R1:4:I.DATA.9   // on clear filtrate P220
                 Lancy_R1:4:I.DATA.10   // Stand by clear filtrate P220
                 Lancy_R1:4:I.DATA.11   // P220 run
                 Lancy_R1:4:I.DATA.12   // clear filtrate flow switch (future)
                 Lancy_R1:4:I.DATA.13   // on cloudy filtrate P230
                 Lancy_R1:4:I.DATA.14   // Stand by cloudy filtrate P230
                 Lancy_R1:4:I.DATA.15   // P230 run
                 Lancy_R1:4:I.POINT_0   // auto filtrate lift station P170
                 Lancy_R1:4:I.POINT_1   // man filtrate lift station P170
                 Lancy_R1:4:I.POINT_2   // P170 run
                 Lancy_R1:4:I.POINT_3   // auto filtrate lift station P180
                 Lancy_R1:4:I.POINT_4   // man filtrate lift station P180
                 Lancy_R1:4:I.POINT_5   // P180 run
                 Lancy_R1:4:I.POINT_6   // on clear filtrate P210
                 Lancy_R1:4:I.POINT_7   // Stand by clear filtrate P210
                 Lancy_R1:4:I.POINT_8   // P210 run
                 Lancy_R1:4:I.POINT_9   // on clear filtrate P220
                 Lancy_R1:4:I.POINT_10   // Stand by clear filtrate P220
                 Lancy_R1:4:I.POINT_11   // P220 run
                 Lancy_R1:4:I.POINT_12   // clear filtrate flow switch (future)
                 Lancy_R1:4:I.POINT_13   // on cloudy filtrate P230
                 Lancy_R1:4:I.POINT_14   // Stand by cloudy filtrate P230
                 Lancy_R1:4:I.POINT_15   // P230 run
            lancy_R1_I6 : vendor 1 type 116 code 12 (SLCChassis 6, rev 1.1, StandardDataDriven RPI 200 ms)
                 Lancy_R1:6:I.DATA.0   // auto L2 filtrate return valve LV325
                 Lancy_R1:6:I.DATA.1   // open L2 filtrate return valve LV325
                 Lancy_R1:6:I.DATA.2   // auto L1 filtrate return valve LV335
                 Lancy_R1:6:I.DATA.3   // open L1 filtrate return valve LV335
                 Lancy_R1:6:I.DATA.4   // auto L3 reactor return valve AV310
                 Lancy_R1:6:I.DATA.5   // close L3 reactor return valve AV310
                 Lancy_R1:6:I.DATA.6   // auto L2 reactor return valve AV320
                 Lancy_R1:6:I.DATA.7   // close L2 reactor return valve AV320
                 Lancy_R1:6:I.DATA.8   // auto L1 reactor return valve AV330
                 Lancy_R1:6:I.DATA.9   // close L1 reactor return valve AV330
                 Lancy_R1:6:I.DATA.10   // surge tank T150 turbidity control
                 Lancy_R1:6:I.DATA.11   // Filtrate lift statio flow switch (future)
                 Lancy_R1:6:I.DATA.12   // M120 overcurrent
                 Lancy_R1:6:I.DATA.13   // P170 overcurrent
                 Lancy_R1:6:I.DATA.14   // P180 overcurrent
                 Lancy_R1:6:I.DATA.15   // P210 overcurrent
                 Lancy_R1:6:I.POINT_0   // auto L2 filtrate return valve LV325
                 Lancy_R1:6:I.POINT_1   // open L2 filtrate return valve LV325
                 Lancy_R1:6:I.POINT_2   // auto L1 filtrate return valve LV335
                 Lancy_R1:6:I.POINT_3   // open L1 filtrate return valve LV335
                 Lancy_R1:6:I.POINT_4   // auto L3 reactor return valve AV310
                 Lancy_R1:6:I.POINT_5   // close L3 reactor return valve AV310
                 Lancy_R1:6:I.POINT_6   // auto L2 reactor return valve AV320
                 Lancy_R1:6:I.POINT_7   // close L2 reactor return valve AV320
                 Lancy_R1:6:I.POINT_8   // auto L1 reactor return valve AV330
                 Lancy_R1:6:I.POINT_9   // close L1 reactor return valve AV330
                 Lancy_R1:6:I.POINT_10   // surge tank T150 turbidity control
                 Lancy_R1:6:I.POINT_11   // Filtrate lift statio flow switch (future)
                 Lancy_R1:6:I.POINT_12   // M120 overcurrent
                 Lancy_R1:6:I.POINT_13   // P170 overcurrent
                 Lancy_R1:6:I.POINT_14   // P180 overcurrent
                 Lancy_R1:6:I.POINT_15   // P210 overcurrent
            lancy_R1_O8 : vendor 1 type 116 code 23 (SLCChassis 8, rev 1.1, StandardDataDriven RPI 200 ms)
                 Lancy_R1:8:O.DATA.0   // filtrate lift pump P170 (20.21.22.886)
                 Lancy_R1:8:O.DATA.1   // P170 run
                 Lancy_R1:8:O.DATA.2   // filtrate lift pump P180 (25,26,27,892)
                 Lancy_R1:8:O.DATA.3   // P180 run
                 Lancy_R1:8:O.DATA.4   // filtrate lift pump seal water valve SV 175
                 Lancy_R1:8:O.DATA.5   // clear filtrate P210 (30,31,32,922)
                 Lancy_R1:8:O.DATA.6   // P210 run
                 Lancy_R1:8:O.DATA.7   // clear filtrate P220 (35,36,67,928)
                 Lancy_R1:8:O.POINT_0   // filtrate lift pump P170 (20.21.22.886)
                 Lancy_R1:8:O.POINT_1   // P170 run
                 Lancy_R1:8:O.POINT_2   // filtrate lift pump P180 (25,26,27,892)
                 Lancy_R1:8:O.POINT_3   // P180 run
                 Lancy_R1:8:O.POINT_4   // filtrate lift pump seal water valve SV 175
                 Lancy_R1:8:O.POINT_5   // clear filtrate P210 (30,31,32,922)
                 Lancy_R1:8:O.POINT_6   // P210 run
                 Lancy_R1:8:O.POINT_7   // clear filtrate P220 (35,36,67,928)
            lancy_R1_I3 : vendor 1 type 116 code 12 (SLCChassis 3, rev 1.1, StandardDataDriven RPI 200 ms)
                 Lancy_R1:3:I.DATA.0   // auto filtrate lift station P170
                 Lancy_R1:3:I.DATA.1   // man filtrate lift station P170
                 Lancy_R1:3:I.DATA.2   // P170 run
                 Lancy_R1:3:I.DATA.3   // auto filtrate lift station P180
                 Lancy_R1:3:I.DATA.4   // man filtrate lift station P180
                 Lancy_R1:3:I.DATA.5   // P180 run
                 Lancy_R1:3:I.DATA.6   // on clear filtrate P210
                 Lancy_R1:3:I.DATA.7   // Stand by clear filtrate P210
                 Lancy_R1:3:I.DATA.8   // P210 run
                 Lancy_R1:3:I.DATA.9   // on clear filtrate P220
                 Lancy_R1:3:I.DATA.10   // Stand by clear filtrate P220
                 Lancy_R1:3:I.DATA.11   // P220 run
                 Lancy_R1:3:I.DATA.12   // clear filtrate flow switch (future)
                 Lancy_R1:3:I.DATA.13   // on cloudy filtrate P230
                 Lancy_R1:3:I.DATA.14   // Stand by cloudy filtrate P230
                 Lancy_R1:3:I.DATA.15   // P230 run
                 Lancy_R1:3:I.POINT_0   // auto filtrate lift station P170
                 Lancy_R1:3:I.POINT_1   // man filtrate lift station P170
                 Lancy_R1:3:I.POINT_2   // P170 run
                 Lancy_R1:3:I.POINT_3   // auto filtrate lift station P180
                 Lancy_R1:3:I.POINT_4   // man filtrate lift station P180
                 Lancy_R1:3:I.POINT_5   // P180 run
                 Lancy_R1:3:I.POINT_6   // on clear filtrate P210
                 Lancy_R1:3:I.POINT_7   // Stand by clear filtrate P210
                 Lancy_R1:3:I.POINT_8   // P210 run
                 Lancy_R1:3:I.POINT_9   // on clear filtrate P220
                 Lancy_R1:3:I.POINT_10   // Stand by clear filtrate P220
                 Lancy_R1:3:I.POINT_11   // P220 run
                 Lancy_R1:3:I.POINT_12   // clear filtrate flow switch (future)
                 Lancy_R1:3:I.POINT_13   // on cloudy filtrate P230
                 Lancy_R1:3:I.POINT_14   // Stand by cloudy filtrate P230
                 Lancy_R1:3:I.POINT_15   // P230 run
            lancy_R1_O9 : vendor 1 type 116 code 23 (SLCChassis 9, rev 1.1, StandardDataDriven RPI 200 ms)
                 Lancy_R1:9:O.DATA.0   // P220 run
                 Lancy_R1:9:O.DATA.1   // clear filtrate seal water valve
                 Lancy_R1:9:O.DATA.2   // cloudy filtrate P230 (40,41,42,936)
                 Lancy_R1:9:O.DATA.3   // P230 run
                 Lancy_R1:9:O.DATA.4   // cloudy filtrate P240 (45,46,47,951)
                 Lancy_R1:9:O.DATA.5   // P240 run
                 Lancy_R1:9:O.DATA.6   // cloudy filtrate seal water valve
                 Lancy_R1:9:O.DATA.7   // vacuum pump P250 pilot relay start (957,676,sp)
                 Lancy_R1:9:O.POINT_0   // P220 run
                 Lancy_R1:9:O.POINT_1   // clear filtrate seal water valve
                 Lancy_R1:9:O.POINT_2   // cloudy filtrate P230 (40,41,42,936)
                 Lancy_R1:9:O.POINT_3   // P230 run
                 Lancy_R1:9:O.POINT_4   // cloudy filtrate P240 (45,46,47,951)
                 Lancy_R1:9:O.POINT_5   // P240 run
                 Lancy_R1:9:O.POINT_6   // cloudy filtrate seal water valve
                 Lancy_R1:9:O.POINT_7   // vacuum pump P250 pilot relay start (957,676,sp)
         arm1_slc2 : vendor 1 type 12 code 228 (Ethernet 192.168.1.3, rev 1.1)
            O16 : vendor 1 type 116 code 30 (SLCChassis 6, rev 1.1, StandardDataDriven RPI 100 ms)
                 arm1_slc2:6:O.DATA.0   // VANNE ALIBERT
                 arm1_slc2:6:O.DATA.1   // VANNE PMP PUITS 1 + IWM
                 arm1_slc2:6:O.DATA.2   // VANNE PMP PUITS 2
                 arm1_slc2:6:O.DATA.4   // RES
                 arm1_slc2:6:O.DATA.5   // RES
                 arm1_slc2:6:O.DATA.6   // RES
                 arm1_slc2:6:O.DATA.7   // RES
                 arm1_slc2:6:O.DATA.8   // RES
                 arm1_slc2:6:O.DATA.9   // L P17 RUN
                 arm1_slc2:6:O.DATA.10   // L P17 STOP/DEF
                 arm1_slc2:6:O.DATA.11   // L PRO 1 STOP/DEF
                 arm1_slc2:6:O.DATA.12   // L P18 STOP/DEF
                 arm1_slc2:6:O.DATA.13   // RES
                 arm1_slc2:6:O.DATA.14   // RES
                 arm1_slc2:6:O.DATA.15   // L PRO 1 RUN
                 arm1_slc2:6:O.DATA.16   // L PRO 1 STOP /DEF
                 arm1_slc2:6:O.DATA.17   // L PRO 2 RUN
                 arm1_slc2:6:O.DATA.18   // L PRO 2 STOP /DEF
                 arm1_slc2:6:O.DATA.19   // L P21 RUN
                 arm1_slc2:6:O.DATA.20   // L P21 STOP/DEF
                 arm1_slc2:6:O.DATA.21   // L P22 RUN
                 arm1_slc2:6:O.DATA.22   // L P22 STOP
                 arm1_slc2:6:O.DATA.23   // L PRO 3 RUN
                 arm1_slc2:6:O.DATA.24   // L PRO 3 STOP
                 arm1_slc2:6:O.DATA.25   // L PMP NETOYAGE P21 REINGINGPMP P21 RUN
                 arm1_slc2:6:O.DATA.26   // L PMP NETOYAGE P21 STOP
                 arm1_slc2:6:O.DATA.27   // L VENTILO S1 RUN
                 arm1_slc2:6:O.DATA.28   // L VENTILO S1 STOP
                 arm1_slc2:6:O.DATA.29   // L P3 RUN
                 arm1_slc2:6:O.DATA.30   // L P3 STOP
                 arm1_slc2:6:O.DATA.31   // L P4 RUN
            O18 : vendor 1 type 116 code 30 (SLCChassis 8, rev 1.1, StandardDataDriven RPI 100 ms)
            O14 : vendor 1 type 116 code 30 (SLCChassis 4, rev 1.1, StandardDataDriven RPI 100 ms)
            O15 : vendor 1 type 116 code 30 (SLCChassis 5, rev 1.1, StandardDataDriven RPI 100 ms)
            I19 : vendor 1 type 116 code 6 (SLCChassis 9, rev 1.1, StandardDataDriven RPI 100 ms)
            O11 : vendor 1 type 116 code 30 (SLCChassis 1, rev 1.1, StandardDataDriven RPI 100 ms)
                 arm1_slc2:1:O.DATA.0   // motor P11 retour L1
                 arm1_slc2:1:O.DATA.1   // P12 Recup L1
                 arm1_slc2:1:O.DATA.2   // P13 Recup L3
                 arm1_slc2:1:O.DATA.3   // P14 Recup L2
                 arm1_slc2:1:O.DATA.4   // P15 Recup L3
                 arm1_slc2:1:O.DATA.5   // P16 RECUP L3
                 arm1_slc2:1:O.DATA.6   // P17 RECUP L4
                 arm1_slc2:1:O.DATA.7   // P18 RECUP L4
                 arm1_slc2:1:O.DATA.8   // PRO 1 OSMOSE MAIN
                 arm1_slc2:1:O.DATA.9   // PRO 1 OSMOSE TRIANGLE
                 arm1_slc2:1:O.DATA.10   // PRO 1 OSMOSE ETOILE
                 arm1_slc2:1:O.DATA.11   // PRO2 OSMOSE MAIN
                 arm1_slc2:1:O.DATA.12   // PRO 2 OSMOSE TRIANGLE
                 arm1_slc2:1:O.DATA.13   // PRO 2 OSMOSE ETOILE
                 arm1_slc2:1:O.DATA.14   // P 21 AZ -> LIJN MAIN
                 arm1_slc2:1:O.DATA.15   // pomp p21 kuip az driehoek P21_KUIP_AZ_DRIE
                 arm1_slc2:1:O.DATA.16   // P 21 AZ -> LIJN TRIANGLE
                 arm1_slc2:1:O.DATA.17   // P 22 AZ -> LIJN MAIN
                 arm1_slc2:1:O.DATA.18   // P 22 AZ -> LIJN ETOILE
                 arm1_slc2:1:O.DATA.19   // P 22 AZ -> LIJN TRIANGLE
                 arm1_slc2:1:O.DATA.20   // PRO 3 OSMOSE MAIN
                 arm1_slc2:1:O.DATA.21   // PRO 3 OSMOSE TRIANGLE
                 arm1_slc2:1:O.DATA.22   // PRO 3 OSMOSE ETOILE
                 arm1_slc2:1:O.DATA.23   // P21 NETTOYAGE MEMMBRANE
                 arm1_slc2:1:O.DATA.24   // VENTILATEUR S1
                 arm1_slc2:1:O.DATA.25   // P3 PRETRAITEE -> USINE MAIN
                 arm1_slc2:1:O.DATA.26   // P3 PRETRAITEE -> USINE DEBLOCAGE
                 arm1_slc2:1:O.DATA.27   // RES
                 arm1_slc2:1:O.DATA.28   // P4 PRETRAITEE -> USINE MAIN
                 arm1_slc2:1:O.DATA.29   // P4 PRETRAITEE -> USINE DEBLOCAGE
                 arm1_slc2:1:O.DATA.30   // RESERVE
                 arm1_slc2:1:O.DATA.31   // P5 RIN9AGE TFB 1.1 ET 1.2
                 arm1_slc2:1:O.POINT_6   // P17
                 arm1_slc2:1:O.POINT_7   // P18
                 arm1_slc2:1:O.POINT_15   // pomp p21 kuip az driehoek P21_KUIP_AZ_DRIE
                 arm1_slc2:1:O.POINT_25   // pomp voeding drive 1 in lijn P3_FAB_LIJN
            O13 : vendor 1 type 116 code 30 (SLCChassis 3, rev 1.1, StandardDataDriven RPI 100 ms)
            O17 : vendor 1 type 116 code 30 (SLCChassis 7, rev 1.1, StandardDataDriven RPI 100 ms)
            O12 : vendor 1 type 116 code 30 (SLCChassis 2, rev 1.1, StandardDataDriven RPI 100 ms)
                 arm1_slc2:2:O.DATA.0   // P6 RIN9AGE TFB 2.1
                 arm1_slc2:2:O.DATA.1   // P23 RECUP KELDER -> STATION
                 arm1_slc2:2:O.DATA.2   // P24 RECUP KELDER -> STATION
                 arm1_slc2:2:O.DATA.3   // AG1 MIXER decanteur neutralisatie
                 arm1_slc2:2:O.DATA.4   // PD3 PMP DOSEUSE ACIDE
                 arm1_slc2:2:O.DATA.5   // PD4 POMPE DOSEUSE ACIDE
                 arm1_slc2:2:O.DATA.6   // PD5 POMPE DOSEUSE SOUDE
                 arm1_slc2:2:O.DATA.7   // PD6 POMPE DOSEUSE SOUDE
                 arm1_slc2:2:O.DATA.8   // AG 2 MIXER VAT FLOCULANT
                 arm1_slc2:2:O.DATA.9   // AG 3 MIXER VAT FLOCULANT
                 arm1_slc2:2:O.DATA.10   // PD7 PMP DOSEUSE FLOCULANT VAT 1
                 arm1_slc2:2:O.DATA.11   // PD8 PMP DOSEUSE FLOCULANT VAT 2
                 arm1_slc2:2:O.DATA.12   // P19 AFVALWATER-> STATION
                 arm1_slc2:2:O.DATA.13   // P20 AFVALWATER-> STATION
         arm1_slc3 : vendor 1 type 12 code 228 (Ethernet 192.168.1.4, rev 1.1)
            NI20 : vendor 1 type 117 code 6 (SLCChassis 1, rev 1.1, StandardDataDriven RPI 100 ms)
            NI22 : vendor 1 type 117 code 6 (SLCChassis 3, rev 1.1, StandardDataDriven RPI 100 ms)
            NI26 : vendor 1 type 117 code 6 (SLCChassis 7, rev 1.1, StandardDataDriven RPI 100 ms)
            NI25 : vendor 1 type 117 code 6 (SLCChassis 6, rev 1.1, StandardDataDriven RPI 100 ms)
            NI23 : vendor 1 type 117 code 6 (SLCChassis 4, rev 1.1, StandardDataDriven RPI 100 ms)
            NI28 : vendor 1 type 117 code 6 (SLCChassis 9, rev 1.1, StandardDataDriven RPI 100 ms)
            NO27 : vendor 1 type 117 code 11 (SLCChassis 8, rev 1.1, StandardDataDriven RPI 100 ms)
            NI21 : vendor 1 type 117 code 6 (SLCChassis 2, rev 1.1, StandardDataDriven RPI 100 ms)
            NI24 : vendor 1 type 117 code 6 (SLCChassis 5, rev 1.1, StandardDataDriven RPI 100 ms)
         arm1_slc1 : vendor 1 type 12 code 228 (Ethernet 192.168.1.2, rev 1.1)
            I2 : vendor 1 type 116 code 6 (SLCChassis 2, rev 1.1, StandardDataDriven RPI 100 ms)
            I7 : vendor 1 type 116 code 6 (SLCChassis 7, rev 1.1, StandardDataDriven RPI 100 ms)
            I9 : vendor 1 type 116 code 6 (SLCChassis 9, rev 1.1, StandardDataDriven RPI 100 ms)
            I10 : vendor 1 type 116 code 6 (SLCChassis 1, rev 1.1, StandardDataDriven RPI 100 ms)
            I6 : vendor 1 type 116 code 6 (SLCChassis 6, rev 1.1, StandardDataDriven RPI 100 ms)
            I8 : vendor 1 type 116 code 6 (SLCChassis 8, rev 1.1, StandardDataDriven RPI 100 ms)
            I3 : vendor 1 type 116 code 6 (SLCChassis 3, rev 1.1, StandardDataDriven RPI 100 ms)
            I5 : vendor 1 type 116 code 6 (SLCChassis 5, rev 1.1, StandardDataDriven RPI 100 ms)
            I4 : vendor 1 type 116 code 6 (SLCChassis 4, rev 1.1, StandardDataDriven RPI 100 ms)
         Ecotech : vendor 1 type 12 code 228 (Ethernet 192.168.1.9, rev 1.1)
            ecotech_o4 : vendor 1 type 116 code 41 (SLCChassis 4, rev 1.1, StandardDataDriven RPI 40 ms)
                 Ecotech:4:O.DATA.0   // T2 product 17 SOL TO L2
                 Ecotech:4:O.DATA.1   // T3 product 18 SOL TO L3
                 Ecotech:4:O.DATA.2   // acid feed pump 1 M
                 Ecotech:4:O.DATA.3   // water feed pump 2 M
                 Ecotech:4:O.DATA.4   // filter feed pump 3 M
                 Ecotech:4:O.DATA.5   // ADD water to APU water tank
                 Ecotech:4:O.DATA.6   // LL acid feed tank alarm light
                 Ecotech:4:O.DATA.7   // LL water feed tank alarm light
                 Ecotech:4:O.DATA.8   // filter water fill light
                 Ecotech:4:O.DATA.9   // filter backwash light
                 Ecotech:4:O.DATA.10   // filter settle light
                 Ecotech:4:O.DATA.11   // APU cycle number 1 CTR
                 Ecotech:4:O.DATA.12   // filter backwash alarm
                 Ecotech:4:O.DATA.13   // cycle time to long alarm
                 Ecotech:4:O.DATA.14   // HL T1 alarm
                 Ecotech:4:O.DATA.15   // LL alarm T1
                 Ecotech:4:O.POINT_0   // T2 product 17 SOL TO L2
                 Ecotech:4:O.POINT_1   // T3 product 18 SOL TO L3
                 Ecotech:4:O.POINT_2   // acid feed pump 1 M
                 Ecotech:4:O.POINT_3   // water feed pump 2 M
                 Ecotech:4:O.POINT_4   // filter feed pump 3 M
                 Ecotech:4:O.POINT_5   // ADD water to APU water tank
                 Ecotech:4:O.POINT_6   // LL acid feed tank alarm light
                 Ecotech:4:O.POINT_7   // LL water feed tank alarm light
                 Ecotech:4:O.POINT_8   // filter water fill light
                 Ecotech:4:O.POINT_9   // filter backwash light
                 Ecotech:4:O.POINT_10   // filter settle light
                 Ecotech:4:O.POINT_11   // APU cycle number 1 CTR
                 Ecotech:4:O.POINT_12   // filter backwash alarm
                 Ecotech:4:O.POINT_13   // cycle time to long alarm
                 Ecotech:4:O.POINT_14   // HL T1 alarm
                 Ecotech:4:O.POINT_15   // LL alarm T1
            ecotech_AI10 : vendor 1 type 117 code 6 (SLCChassis 10, rev 1.1, StandardDataDriven RPI 40 ms)
                 Ecotech:10:I.CHANNEL_0_DATA   // arrivée air comprimé
                 Ecotech:10:I.CHANNEL_1_DATA   // condfuctivité 4 ma 0 mS 20 ma 300 mS
                 Ecotech:10:I.CHANNEL_2_DATA   // niveau APU feed tank
                 Ecotech:10:I.CHANNEL_3_DATA   // niveau filter feed tank
                 Ecotech:10:I.CHANNEL_4_DATA   // niveau Water APU feed Tank
                 Ecotech:10:I.CHANNEL_5_DATA   // RESERVE
                 Ecotech:10:I.CHANNEL_6_DATA   // RESERVE
                 Ecotech:10:I.CHANNEL_7_DATA   // RESERVE
            ecotech_i8 : vendor 1 type 116 code 4 (SLCChassis 8, rev 1.1, StandardDataDriven RPI 40 ms)
                 Ecotech:8:I.DATA.0   // tank 4 selected
                 Ecotech:8:I.DATA.1   // HL tank A
                 Ecotech:8:I.DATA.2   // LL tank A
                 Ecotech:8:I.DATA.3   // HL tank B
                 Ecotech:8:I.DATA.4   // LL tank B
                 Ecotech:8:I.DATA.5   // lijn 4 working
                 Ecotech:8:I.DATA.6   // RESERVE
                 Ecotech:8:I.DATA.7   // RESERVE
            ecotech_i7 : vendor 1 type 116 code 4 (SLCChassis 7, rev 1.1, StandardDataDriven RPI 40 ms)
                 Ecotech:7:I.DATA.0   // filter feed LL
                 Ecotech:7:I.DATA.1   // filter feed HL
                 Ecotech:7:I.DATA.2   // HL APU water tank
                 Ecotech:7:I.DATA.3   // LL APU water tank
                 Ecotech:7:I.DATA.4   // LL APU feed tank
                 Ecotech:7:I.DATA.5   // HL alarm APU feed tank
                 Ecotech:7:I.DATA.6   // bp manual count reset
                 Ecotech:7:I.DATA.7   // RESERVE
                 Ecotech:7:I.POINT_0   // filter feed LL
                 Ecotech:7:I.POINT_1   // filter feed HL
                 Ecotech:7:I.POINT_2   // HL APU water tank
                 Ecotech:7:I.POINT_3   // LL APU water tank
                 Ecotech:7:I.POINT_4   // LL APU feed tank
                 Ecotech:7:I.POINT_5   // HL alarm APU feed tank
                 Ecotech:7:I.POINT_6   // bp manual count reset
                 Ecotech:7:I.POINT_7   // RESERVE
            ecotech_o6 : vendor 1 type 116 code 40 (SLCChassis 6, rev 1.1, StandardDataDriven RPI 40 ms)
                 Ecotech:6:O.DATA.0   // onstream light
                 Ecotech:6:O.DATA.1   // RESERVE
                 Ecotech:6:O.DATA.2   // acid inlet 1 SOL
                 Ecotech:6:O.DATA.3   // RESERVE
                 Ecotech:6:O.DATA.4   // manual count reset
                 Ecotech:6:O.DATA.5   // RESERVE
                 Ecotech:6:O.DATA.6   // RESERVE
                 Ecotech:6:O.DATA.7   // RESERVE
                 Ecotech:6:O.POINT_0   // onstream light
                 Ecotech:6:O.POINT_1   // RESERVE
                 Ecotech:6:O.POINT_2   // acid inlet 1 SOL
                 Ecotech:6:O.POINT_3   // RESERVE
                 Ecotech:6:O.POINT_4   // manual count reset
                 Ecotech:6:O.POINT_5   // RESERVE
                 Ecotech:6:O.POINT_6   // RESERVE
                 Ecotech:6:O.POINT_7   // RESERVE
            ecotech_o3 : vendor 1 type 116 code 41 (SLCChassis 3, rev 1.1, StandardDataDriven RPI 40 ms)
                 Ecotech:3:O.DATA.0   // RESERVE
                 Ecotech:3:O.DATA.1   // water inlet 2 SOL
                 Ecotech:3:O.DATA.2   // water displ void 3 SOL
                 Ecotech:3:O.DATA.3   // by-product 4 SOL
                 Ecotech:3:O.DATA.4   // product 5 SOL
                 Ecotech:3:O.DATA.5   // acid displ void 6 SOL
                 Ecotech:3:O.DATA.6   // filter feed inlet 7 SOL
                 Ecotech:3:O.DATA.7   // filter top air inlet 8 SOL
                 Ecotech:3:O.DATA.8   // filter top waste outlet 9 SOL
                 Ecotech:3:O.DATA.9   // filter bottom waste outlet 10 SOL
                 Ecotech:3:O.DATA.10   // filter bottom air inlet 11 SOL
                 Ecotech:3:O.DATA.11   // bottom outlet to feed tank
                 Ecotech:3:O.DATA.12   // filter outlet to feed tank 13 SOL
                 Ecotech:3:O.DATA.13   // filter water inlet 14 SOL
                 Ecotech:3:O.DATA.14   // filter filtered outlet 15 SOL
                 Ecotech:3:O.DATA.15   // T1 product 16 SOL TO L1
                 Ecotech:3:O.POINT_1   // water inlet 2 SOL
                 Ecotech:3:O.POINT_2   // water displ void 3 SOL
                 Ecotech:3:O.POINT_3   // by-product 4 SOL
                 Ecotech:3:O.POINT_4   // product 5 SOL
                 Ecotech:3:O.POINT_5   // acid displ void 6 SOL
                 Ecotech:3:O.POINT_6   // filter feed inlet 7 SOL
                 Ecotech:3:O.POINT_7   // filter top air inlet 8 SOL
                 Ecotech:3:O.POINT_8   // filter top waste outlet 9 SOL
                 Ecotech:3:O.POINT_9   // filter bottom waste outlet 10 SOL
                 Ecotech:3:O.POINT_10   // filter bottom air inlet 11 SOL
                 Ecotech:3:O.POINT_11   // bottom outlet to feed tank
                 Ecotech:3:O.POINT_12   // filter outlet to feed tank 13 SOL
                 Ecotech:3:O.POINT_13   // filter water inlet 14 SOL
                 Ecotech:3:O.POINT_14   // filter filtered outlet 15 SOL
                 Ecotech:3:O.POINT_15   // T1 product 16 SOL TO L1
            ecotech_o9 : vendor 1 type 116 code 27 (SLCChassis 9, rev 1.1, StandardDataDriven RPI 40 ms)
                 Ecotech:9:O.DATA.0   // APU feed van lijn
                 Ecotech:9:O.DATA.1   // APU product naar lijn 4
                 Ecotech:9:O.DATA.2   // HL alarm tank 4
                 Ecotech:9:O.DATA.3   // LL alarm tank 4
                 Ecotech:9:O.DATA.4   // tank 4 selected
                 Ecotech:9:O.DATA.5   // RESERVE
                 Ecotech:9:O.DATA.6   // RESERVE
                 Ecotech:9:O.DATA.7   // RESERVE
                 Ecotech:9:O.POINT_0   // APU feed van lijn
                 Ecotech:9:O.POINT_1   // APU product naar lijn 4
                 Ecotech:9:O.POINT_2   // HL alarm tank 4
                 Ecotech:9:O.POINT_3   // LL alarm tank 4
                 Ecotech:9:O.POINT_4   // tank 4 selected
                 Ecotech:9:O.POINT_5   // RESERVE
                 Ecotech:9:O.POINT_6   // RESERVE
                 Ecotech:9:O.POINT_7   // RESERVE
            ecotech_i1 : vendor 1 type 116 code 5 (SLCChassis 1, rev 1.1, StandardDataDriven RPI 20 ms)
                 Ecotech:1:I.DATA.0   // shutdown run switch
                 Ecotech:1:I.DATA.1   // volumetric pulser
                 Ecotech:1:I.DATA.2   // T1 selected
                 Ecotech:1:I.DATA.3   // T2 selected
                 Ecotech:1:I.DATA.4   // T3 selected
                 Ecotech:1:I.DATA.5   // HL APU feed tank
                 Ecotech:1:I.DATA.6   // LL APU feed tank
                 Ecotech:1:I.DATA.7   // HL water tank
                 Ecotech:1:I.DATA.8   // LL water tank
                 Ecotech:1:I.DATA.9   // HL filter feed tank
                 Ecotech:1:I.DATA.10   // LL filter feed tank
                 Ecotech:1:I.DATA.11   // HL T1
                 Ecotech:1:I.DATA.12   // LL T1
                 Ecotech:1:I.DATA.13   // alarm silence buttom 3 PB
                 Ecotech:1:I.DATA.14   // filter float switch
                 Ecotech:1:I.DATA.15   // filter backwash initiate button
                 Ecotech:1:I.POINT_0   // shutdown run switch
                 Ecotech:1:I.POINT_1   // volumetric pulser
                 Ecotech:1:I.POINT_2   // T1 selected
                 Ecotech:1:I.POINT_3   // T2 selected
                 Ecotech:1:I.POINT_4   // T3 selected
                 Ecotech:1:I.POINT_5   // HL APU feed tank
                 Ecotech:1:I.POINT_6   // LL APU feed tank
                 Ecotech:1:I.POINT_7   // HL water tank
                 Ecotech:1:I.POINT_8   // LL water tank
                 Ecotech:1:I.POINT_9   // HL filter feed tank
                 Ecotech:1:I.POINT_10   // LL filter feed tank
                 Ecotech:1:I.POINT_11   // HL T1
                 Ecotech:1:I.POINT_12   // LL T1
                 Ecotech:1:I.POINT_13   // alarm silence buttom 3 PB
                 Ecotech:1:I.POINT_14   // filter float switch
                 Ecotech:1:I.POINT_15   // filter backwash initiate button
            ecotech_i2 : vendor 1 type 116 code 5 (SLCChassis 2, rev 1.1, StandardDataDriven RPI 400 ms)
                 Ecotech:2:I.DATA.0   // HL T2
                 Ecotech:2:I.DATA.1   // LL T2
                 Ecotech:2:I.DATA.2   // HL T3
                 Ecotech:2:I.DATA.3   // LL T3
                 Ecotech:2:I.DATA.4   // RESERVE
                 Ecotech:2:I.DATA.5   // RESERVE
                 Ecotech:2:I.DATA.6   // RESERVE
                 Ecotech:2:I.DATA.7   // RESERVE
                 Ecotech:2:I.DATA.8   // L flow filter feed pump
                 Ecotech:2:I.DATA.9   // presure switch
                 Ecotech:2:I.DATA.10   // L flow APU feed pump
                 Ecotech:2:I.DATA.11   // L flow APU water pump
                 Ecotech:2:I.DATA.12   // overload APU feed pump
                 Ecotech:2:I.DATA.13   // overload water pump
                 Ecotech:2:I.DATA.14   // overload filter feed pump
                 Ecotech:2:I.DATA.15   // RESERVE
                 Ecotech:2:I.POINT_0   // HL T2
                 Ecotech:2:I.POINT_1   // LL T2
                 Ecotech:2:I.POINT_2   // HL T3
                 Ecotech:2:I.POINT_3   // LL T3
                 Ecotech:2:I.POINT_4   // RESERVE
                 Ecotech:2:I.POINT_5   // RESERVE
                 Ecotech:2:I.POINT_6   // RESERVE
                 Ecotech:2:I.POINT_7   // RESERVE
                 Ecotech:2:I.POINT_8   // L flow filter feed pump
                 Ecotech:2:I.POINT_9   // presure switch
                 Ecotech:2:I.POINT_10   // L flow APU feed pump
                 Ecotech:2:I.POINT_11   // L flow APU water pump
                 Ecotech:2:I.POINT_12   // overload APU feed pump
                 Ecotech:2:I.POINT_13   // overload water pump
                 Ecotech:2:I.POINT_14   // overload filter feed pump
                 Ecotech:2:I.POINT_15   // RESERVE
            ecotech_o5 : vendor 1 type 116 code 41 (SLCChassis 5, rev 1.1, StandardDataDriven RPI 40 ms)
                 Ecotech:5:O.DATA.0   // HL alarm T2
                 Ecotech:5:O.DATA.1   // LL alarm T2
                 Ecotech:5:O.DATA.2   // HL alarm T3
                 Ecotech:5:O.DATA.3   // LL alarm T3
                 Ecotech:5:O.DATA.4   // L flow filter feed pump
                 Ecotech:5:O.DATA.5   // cycle in proces light
                 Ecotech:5:O.DATA.6   // cycle conpleted light
                 Ecotech:5:O.DATA.7   // filter sweeten off
                 Ecotech:5:O.DATA.8   // T1 transfer OK 19 SOL from L1
                 Ecotech:5:O.DATA.9   // T2 transfer OK 20 SOL FROM L2
                 Ecotech:5:O.DATA.10   // T3 transfer OK 21 SOL FROM L3
                 Ecotech:5:O.DATA.11   // L flow APU feed pump alarm
                 Ecotech:5:O.DATA.12   // L flow APU water pump alarm
                 Ecotech:5:O.DATA.13   // overload APU feed pump alarm
                 Ecotech:5:O.DATA.14   // overload water pump alarm
                 Ecotech:5:O.DATA.15   // filter feed pump overload alarm
                 Ecotech:5:O.POINT_0   // HL alarm T2
                 Ecotech:5:O.POINT_1   // LL alarm T2
                 Ecotech:5:O.POINT_2   // HL alarm T3
                 Ecotech:5:O.POINT_3   // LL alarm T3
                 Ecotech:5:O.POINT_4   // L flow filter feed pump
                 Ecotech:5:O.POINT_5   // cycle in proces light
                 Ecotech:5:O.POINT_6   // cycle conpleted light
                 Ecotech:5:O.POINT_7   // filter sweeten off
                 Ecotech:5:O.POINT_8   // T1 transfer OK 19 SOL from L1
                 Ecotech:5:O.POINT_9   // T2 transfer OK 20 SOL FROM L2
                 Ecotech:5:O.POINT_10   // T3 transfer OK 21 SOL FROM L3
                 Ecotech:5:O.POINT_11   // L flow APU feed pump alarm
                 Ecotech:5:O.POINT_12   // L flow APU water pump alarm
                 Ecotech:5:O.POINT_13   // overload APU feed pump alarm
                 Ecotech:5:O.POINT_14   // overload water pump alarm
                 Ecotech:5:O.POINT_15   // filter feed pump overload alarm
END_MODULES
